// Mitsubishi GX Works2 project: 미쯔비시   PLC: Q02U

PROGRAM INPUT
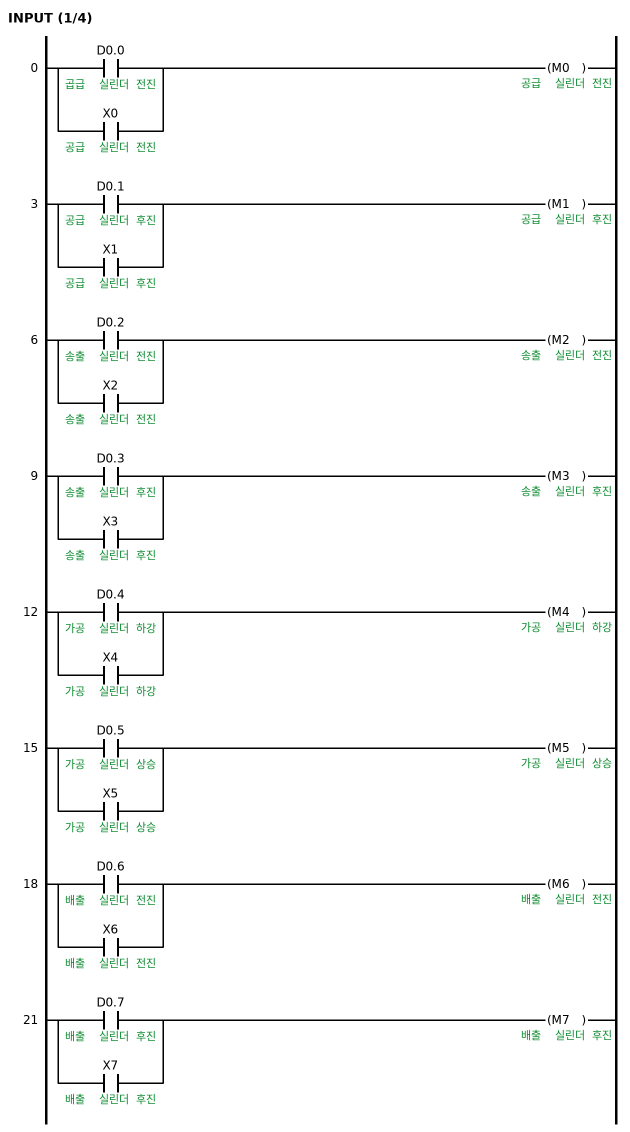
0     LD      D0.0  ; 곱급    실린더  전진
      OR      X0  ; 공급    실린더  전진
      OUT     M0  ; 공급    실린더  전진
3     LD      D0.1  ; 공급    실린더  후진
      OR      X1  ; 공급    실린더  후진
      OUT     M1  ; 공급    실린더  후진
6     LD      D0.2  ; 송출    실린더  전진
      OR      X2  ; 송출    실린더  전진
      OUT     M2  ; 송출    실린더  전진
9     LD      D0.3  ; 송출    실린더  후진
      OR      X3  ; 송출    실린더  후진
      OUT     M3  ; 송출    실린더  후진
12    LD      D0.4  ; 가공    실린더  하강
      OR      X4  ; 가공    실린더  하강
      OUT     M4  ; 가공    실린더  하강
15    LD      D0.5  ; 가공    실린더  상승
      OR      X5  ; 가공    실린더  상승
      OUT     M5  ; 가공    실린더  상승
18    LD      D0.6  ; 배출    실린더  전진
      OR      X6  ; 배출    실린더  전진
      OUT     M6  ; 배출    실린더  전진
21    LD      D0.7  ; 배출    실린더  후진
      OR      X7  ; 배출    실린더  후진
      OUT     M7  ; 배출    실린더  후진
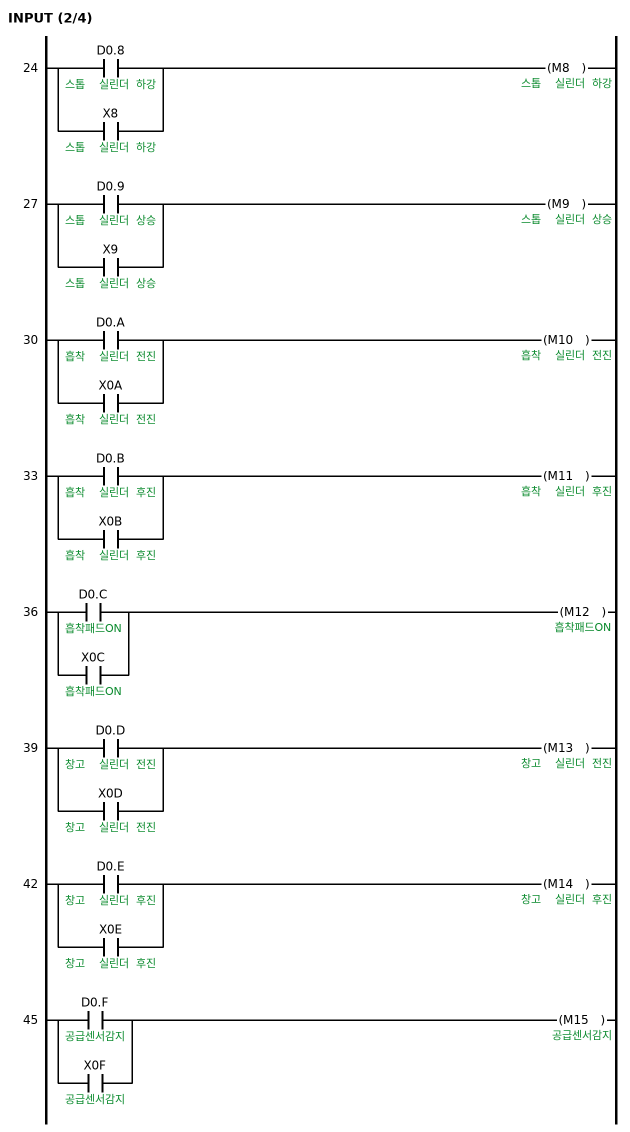
24    LD      D0.8  ; 스톱    실린더  하강
      OR      X8  ; 스톱    실린더  하강
      OUT     M8  ; 스톱    실린더  하강
27    LD      D0.9  ; 스톱    실린더  상승
      OR      X9  ; 스톱    실린더  상승
      OUT     M9  ; 스톱    실린더  상승
30    LD      D0.A  ; 흡착    실린더  전진
      OR      X0A  ; 흡착    실린더  전진
      OUT     M10  ; 흡착    실린더  전진
33    LD      D0.B  ; 흡착    실린더  후진
      OR      X0B  ; 흡착    실린더  후진
      OUT     M11  ; 흡착    실린더  후진
36    LD      D0.C  ; 흡착패드ON
      OR      X0C  ; 흡착패드ON
      OUT     M12  ; 흡착패드ON
39    LD      D0.D  ; 창고    실린더  전진
      OR      X0D  ; 창고    실린더  전진
      OUT     M13  ; 창고    실린더  전진
42    LD      D0.E  ; 창고    실린더  후진
      OR      X0E  ; 창고    실린더  후진
      OUT     M14  ; 창고    실린더  후진
45    LD      D0.F  ; 공급센서감지
      OR      X0F  ; 공급센서감지
      OUT     M15  ; 공급센서감지
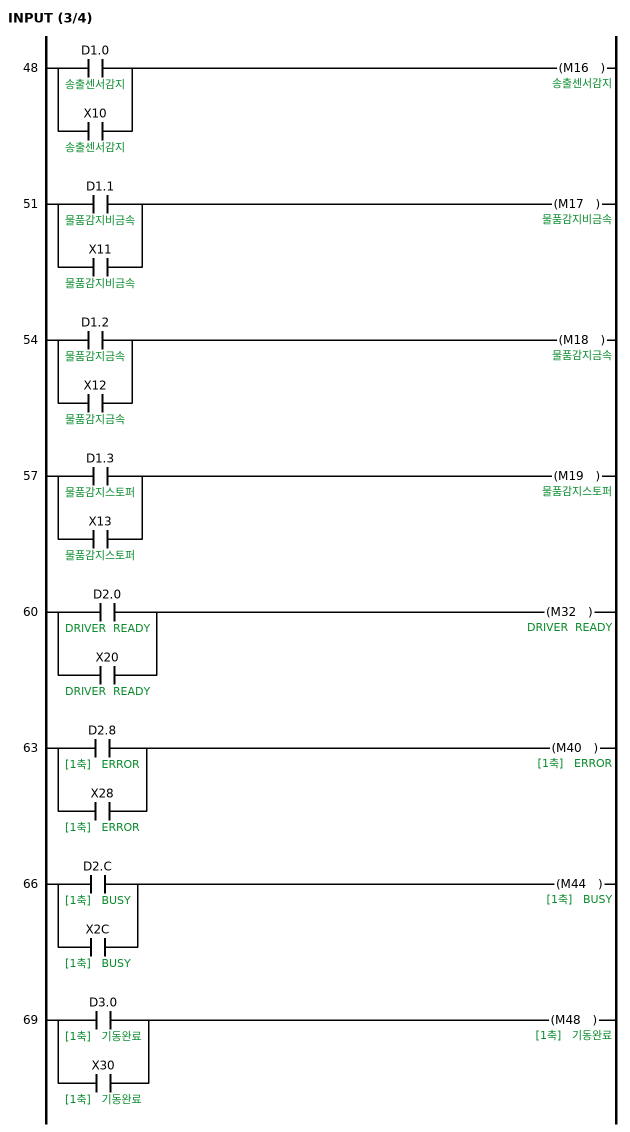
48    LD      D1.0  ; 송출센서감지
      OR      X10  ; 송출센서감지
      OUT     M16  ; 송출센서감지
51    LD      D1.1  ; 물품감지비금속
      OR      X11  ; 물품감지비금속
      OUT     M17  ; 물품감지비금속
54    LD      D1.2  ; 물품감지금속
      OR      X12  ; 물품감지금속
      OUT     M18  ; 물품감지금속
57    LD      D1.3  ; 물품감지스토퍼
      OR      X13  ; 물품감지스토퍼
      OUT     M19  ; 물품감지스토퍼
60    LD      D2.0  ; DRIVER  READY
      OR      X20  ; DRIVER  READY
      OUT     M32  ; DRIVER  READY
63    LD      D2.8  ; [1축]   ERROR
      OR      X28  ; [1축]   ERROR
      OUT     M40  ; [1축]   ERROR
66    LD      D2.C  ; [1축]   BUSY
      OR      X2C  ; [1축]   BUSY
      OUT     M44  ; [1축]   BUSY
69    LD      D3.0  ; [1축]   기동완료
      OR      X30  ; [1축]   기동완료
      OUT     M48  ; [1축]   기동완료
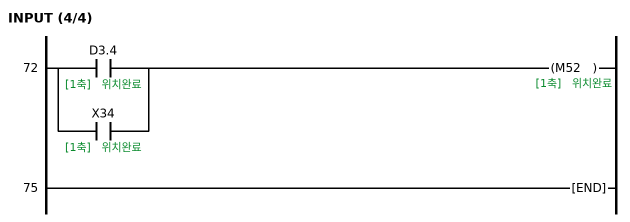
72    LD      D3.4  ; [1축]   위치완료
      OR      X34  ; [1축]   위치완료
      OUT     M52  ; [1축]   위치완료
75    END
END_PROGRAM

PROGRAM OUTPUT
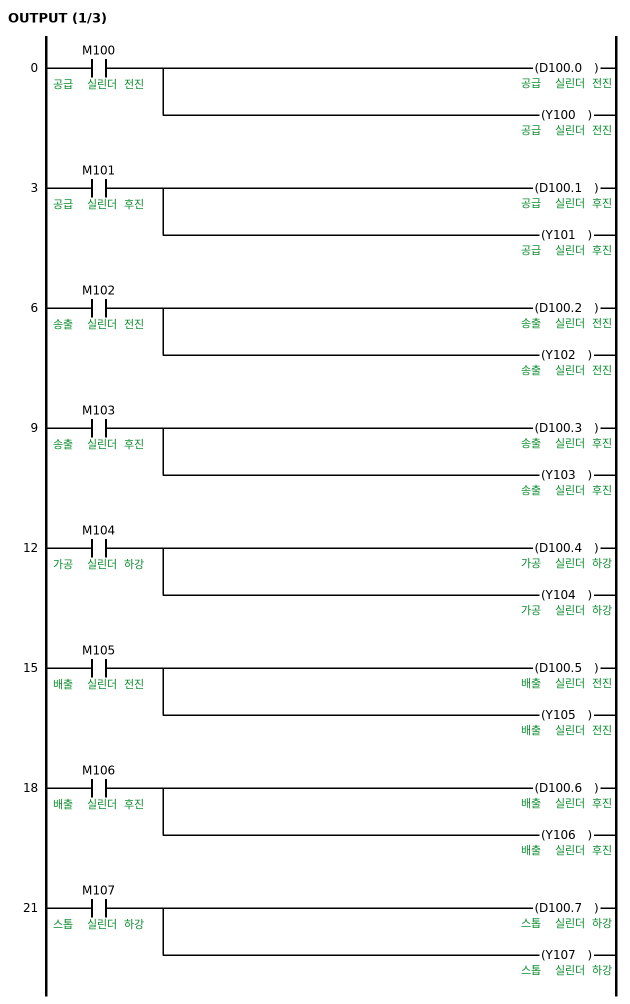
0     LD      M100  ; 공급    실린더  전진
      OUT     D100.0  ; 공급    실린더  전진
      OUT     Y100  ; 공급    실린더  전진
3     LD      M101  ; 공급    실린더  후진
      OUT     D100.1  ; 공급    실린더  후진
      OUT     Y101  ; 공급    실린더  후진
6     LD      M102  ; 송출    실린더  전진
      OUT     D100.2  ; 송출    실린더  전진
      OUT     Y102  ; 송출    실린더  전진
9     LD      M103  ; 송출    실린더  후진
      OUT     D100.3  ; 송출    실린더  후진
      OUT     Y103  ; 송출    실린더  후진
12    LD      M104  ; 가공    실린더  하강
      OUT     D100.4  ; 가공    실린더  하강
      OUT     Y104  ; 가공    실린더  하강
15    LD      M105  ; 배출    실린더  전진
      OUT     D100.5  ; 배출    실린더  전진
      OUT     Y105  ; 배출    실린더  전진
18    LD      M106  ; 배출    실린더  후진
      OUT     D100.6  ; 배출    실린더  후진
      OUT     Y106  ; 배출    실린더  후진
21    LD      M107  ; 스톱    실린더  하강
      OUT     D100.7  ; 스톱    실린더  하강
      OUT     Y107  ; 스톱    실린더  하강
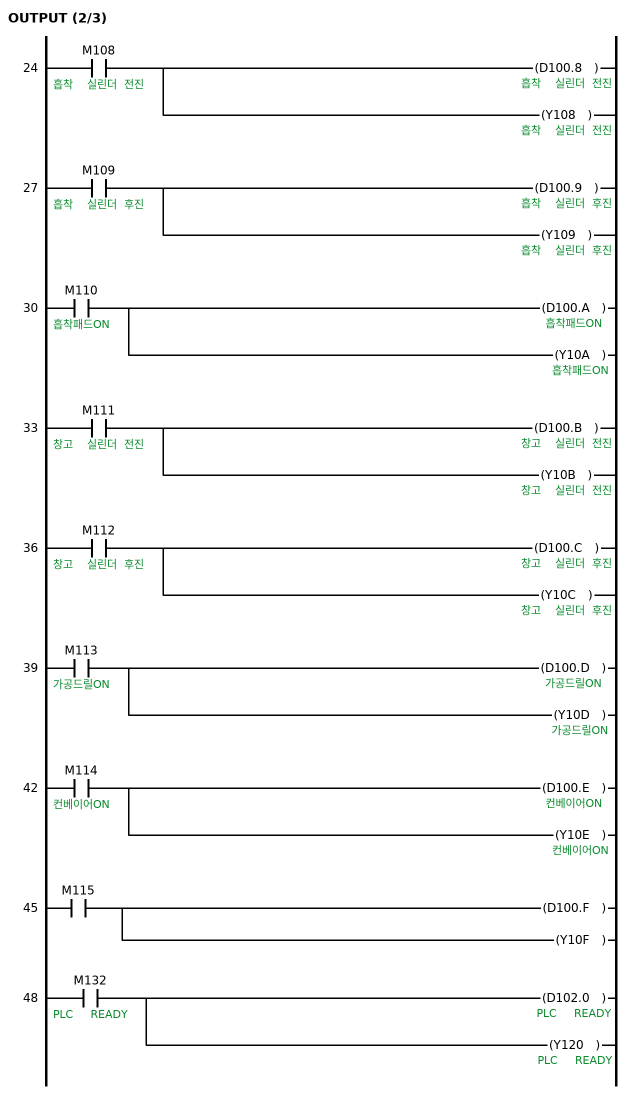
24    LD      M108  ; 흡착    실린더  전진
      OUT     D100.8  ; 흡착    실린더  전진
      OUT     Y108  ; 흡착    실린더  전진
27    LD      M109  ; 흡착    실린더  후진
      OUT     D100.9  ; 흡착    실린더  후진
      OUT     Y109  ; 흡착    실린더  후진
30    LD      M110  ; 흡착패드ON
      OUT     D100.A  ; 흡착패드ON
      OUT     Y10A  ; 흡착패드ON
33    LD      M111  ; 창고    실린더  전진
      OUT     D100.B  ; 창고    실린더  전진
      OUT     Y10B  ; 창고    실린더  전진
36    LD      M112  ; 창고    실린더  후진
      OUT     D100.C  ; 창고    실린더  후진
      OUT     Y10C  ; 창고    실린더  후진
39    LD      M113  ; 가공드릴ON
      OUT     D100.D  ; 가공드릴ON
      OUT     Y10D  ; 가공드릴ON
42    LD      M114  ; 컨베이어ON
      OUT     D100.E  ; 컨베이어ON
      OUT     Y10E  ; 컨베이어ON
45    LD      M115
      OUT     D100.F
      OUT     Y10F
48    LD      M132  ; PLC     READY
      OUT     D102.0  ; PLC     READY
      OUT     Y120  ; PLC     READY
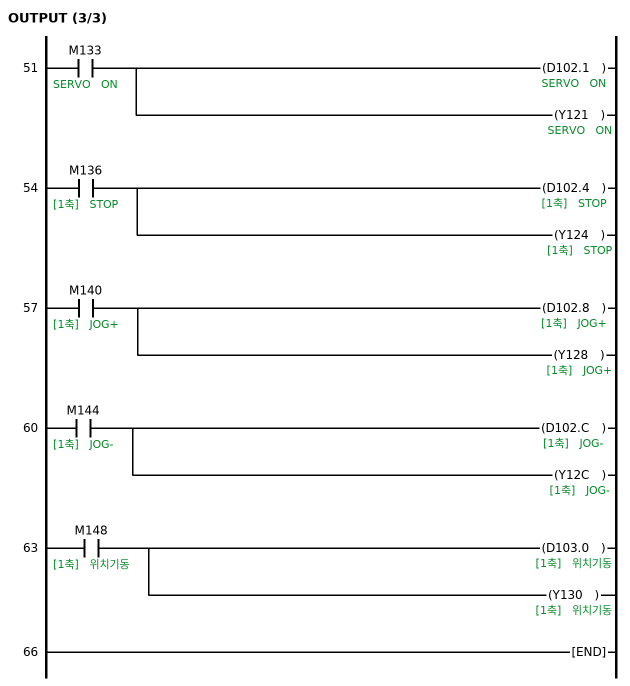
51    LD      M133  ; SERVO   ON
      OUT     D102.1  ; SERVO   ON
      OUT     Y121  ; SERVO   ON
54    LD      M136  ; [1축]   STOP
      OUT     D102.4  ; [1축]   STOP
      OUT     Y124  ; [1축]   STOP
57    LD      M140  ; [1축]   JOG+
      OUT     D102.8  ; [1축]   JOG+
      OUT     Y128  ; [1축]   JOG+
60    LD      M144  ; [1축]   JOG-
      OUT     D102.C  ; [1축]   JOG-
      OUT     Y12C  ; [1축]   JOG-
63    LD      M148  ; [1축]   위치기동
      OUT     D103.0  ; [1축]   위치기동
      OUT     Y130  ; [1축]   위치기동
66    END
END_PROGRAM

PROGRAM CONTROL
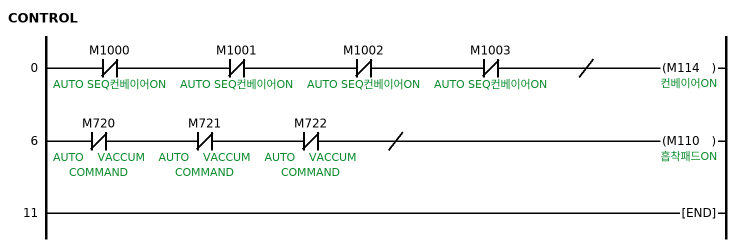
0     LDI     M1000  ; AUTO SEQ컨베이어ON
      ANI     M1001  ; AUTO SEQ컨베이어ON
      ANI     M1002  ; AUTO SEQ컨베이어ON
      ANI     M1003  ; AUTO SEQ컨베이어ON
      INV
      OUT     M114  ; 컨베이어ON
6     LDI     M720  ; AUTO    VACCUM  COMMAND
      ANI     M721  ; AUTO    VACCUM  COMMAND
      ANI     M722  ; AUTO    VACCUM  COMMAND
      INV
      OUT     M110  ; 흡착패드ON
11    END
END_PROGRAM

PROGRAM SUPPLY
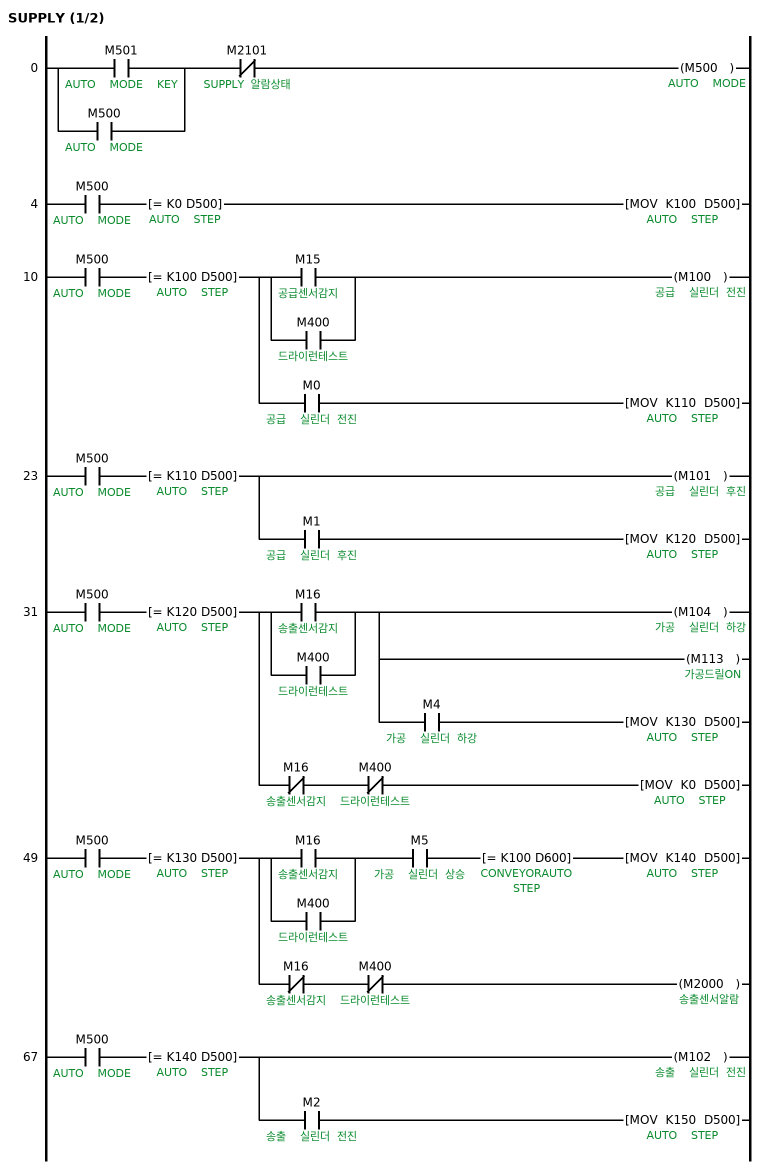
0     LD      M501  ; AUTO    MODE    KEY
      OR      M500  ; AUTO    MODE
      ANI     M2101  ; SUPPLY  알람상태
      OUT     M500  ; AUTO    MODE
4     LD      M500  ; AUTO    MODE
      AND=    K0 D500  ; AUTO    STEP
      MOV     K100 D500
10    LD      M500  ; AUTO    MODE
      AND=    K100 D500  ; AUTO    STEP
      MPS
      LD      M15  ; 공급센서감지
      OR      M400  ; 드라이런테스트
      ANB
      OUT     M100  ; 공급    실린더  전진
      MPP
      AND     M0  ; 공급    실린더  전진
      MOV     K110 D500
23    LD      M500  ; AUTO    MODE
      AND=    K110 D500  ; AUTO    STEP
      OUT     M101  ; 공급    실린더  후진
      AND     M1  ; 공급    실린더  후진
      MOV     K120 D500
31    LD      M500  ; AUTO    MODE
      AND=    K120 D500  ; AUTO    STEP
      MPS
      LD      M16  ; 송출센서감지
      OR      M400  ; 드라이런테스트
      ANB
      OUT     M104  ; 가공    실린더  하강
      OUT     M113  ; 가공드릴ON
      AND     M4  ; 가공    실린더  하강
      MOV     K130 D500
      MPP
      ANI     M16  ; 송출센서감지
      ANI     M400  ; 드라이런테스트
      MOV     K0 D500
49    LD      M500  ; AUTO    MODE
      AND=    K130 D500  ; AUTO    STEP
      MPS
      LD      M16  ; 송출센서감지
      OR      M400  ; 드라이런테스트
      ANB
      AND     M5  ; 가공    실린더  상승
      AND=    K100 D600  ; CONVEYORAUTO    STEP
      MOV     K140 D500
      MPP
      ANI     M16  ; 송출센서감지
      ANI     M400  ; 드라이런테스트
      OUT     M2000  ; 송출센서알람
67    LD      M500  ; AUTO    MODE
      AND=    K140 D500  ; AUTO    STEP
      OUT     M102  ; 송출    실린더  전진
      AND     M2  ; 송출    실린더  전진
      MOV     K150 D500
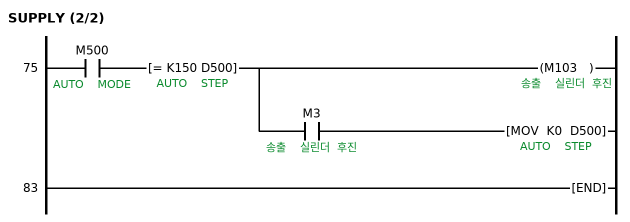
75    LD      M500  ; AUTO    MODE
      AND=    K150 D500  ; AUTO    STEP
      OUT     M103  ; 송출    실린더  후진
      AND     M3  ; 송출    실린더  후진
      MOV     K0 D500
83    END
END_PROGRAM

PROGRAM CONVEYOR
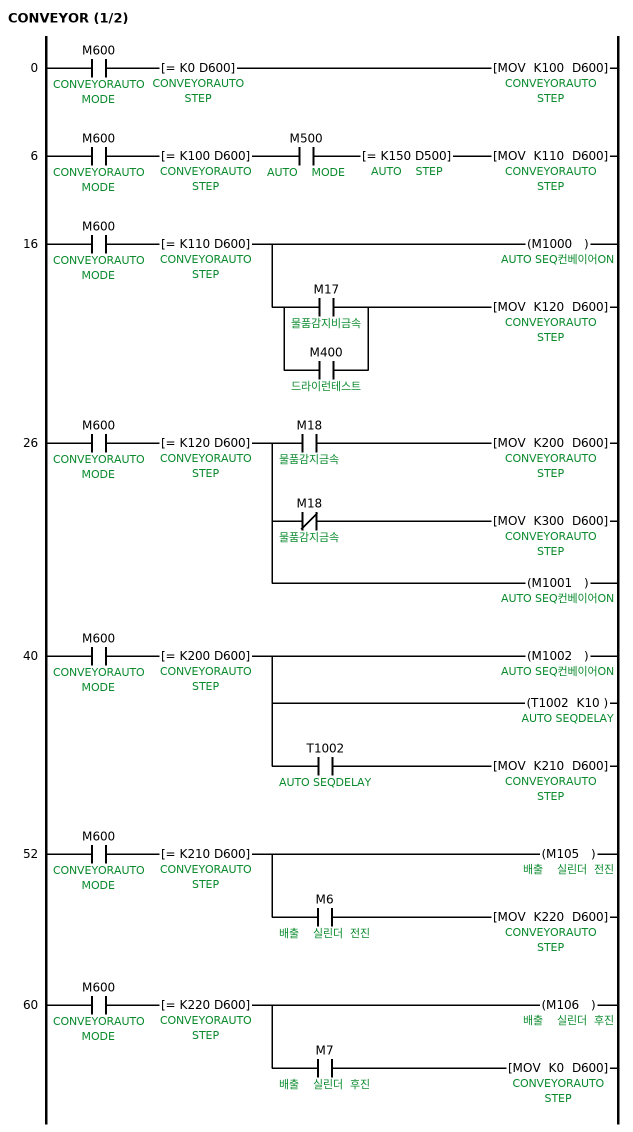
0     LD      M600  ; CONVEYORAUTO    MODE
      AND=    K0 D600  ; CONVEYORAUTO    STEP
      MOV     K100 D600
6     LD      M600  ; CONVEYORAUTO    MODE
      AND=    K100 D600  ; CONVEYORAUTO    STEP
      AND     M500  ; AUTO    MODE
      AND=    K150 D500  ; AUTO    STEP
      MOV     K110 D600
16    LD      M600  ; CONVEYORAUTO    MODE
      AND=    K110 D600  ; CONVEYORAUTO    STEP
      OUT     M1000  ; AUTO SEQ컨베이어ON
      LD      M17  ; 물품감지비금속
      OR      M400  ; 드라이런테스트
      ANB
      MOV     K120 D600
26    LD      M600  ; CONVEYORAUTO    MODE
      AND=    K120 D600  ; CONVEYORAUTO    STEP
      MPS
      AND     M18  ; 물품감지금속
      MOV     K200 D600
      MRD
      ANI     M18  ; 물품감지금속
      MOV     K300 D600
      MPP
      OUT     M1001  ; AUTO SEQ컨베이어ON
40    LD      M600  ; CONVEYORAUTO    MODE
      AND=    K200 D600  ; CONVEYORAUTO    STEP
      OUT     M1002  ; AUTO SEQ컨베이어ON
      OUT     T1002 K10  ; AUTO SEQDELAY
      AND     T1002  ; AUTO SEQDELAY
      MOV     K210 D600
52    LD      M600  ; CONVEYORAUTO    MODE
      AND=    K210 D600  ; CONVEYORAUTO    STEP
      OUT     M105  ; 배출    실린더  전진
      AND     M6  ; 배출    실린더  전진
      MOV     K220 D600
60    LD      M600  ; CONVEYORAUTO    MODE
      AND=    K220 D600  ; CONVEYORAUTO    STEP
      OUT     M106  ; 배출    실린더  후진
      AND     M7  ; 배출    실린더  후진
      MOV     K0 D600
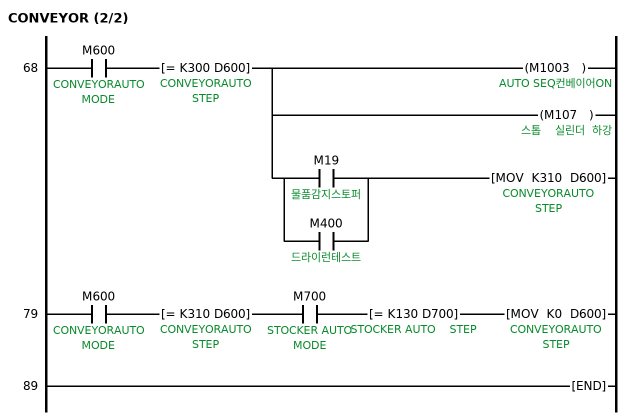
68    LD      M600  ; CONVEYORAUTO    MODE
      AND=    K300 D600  ; CONVEYORAUTO    STEP
      OUT     M1003  ; AUTO SEQ컨베이어ON
      OUT     M107  ; 스톱    실린더  하강
      LD      M19  ; 물품감지스토퍼
      OR      M400  ; 드라이런테스트
      ANB
      MOV     K310 D600
79    LD      M600  ; CONVEYORAUTO    MODE
      AND=    K310 D600  ; CONVEYORAUTO    STEP
      AND     M700  ; STOCKER AUTO    MODE
      AND=    K130 D700  ; STOCKER AUTO    STEP
      MOV     K0 D600
89    END
END_PROGRAM

PROGRAM STOCKER
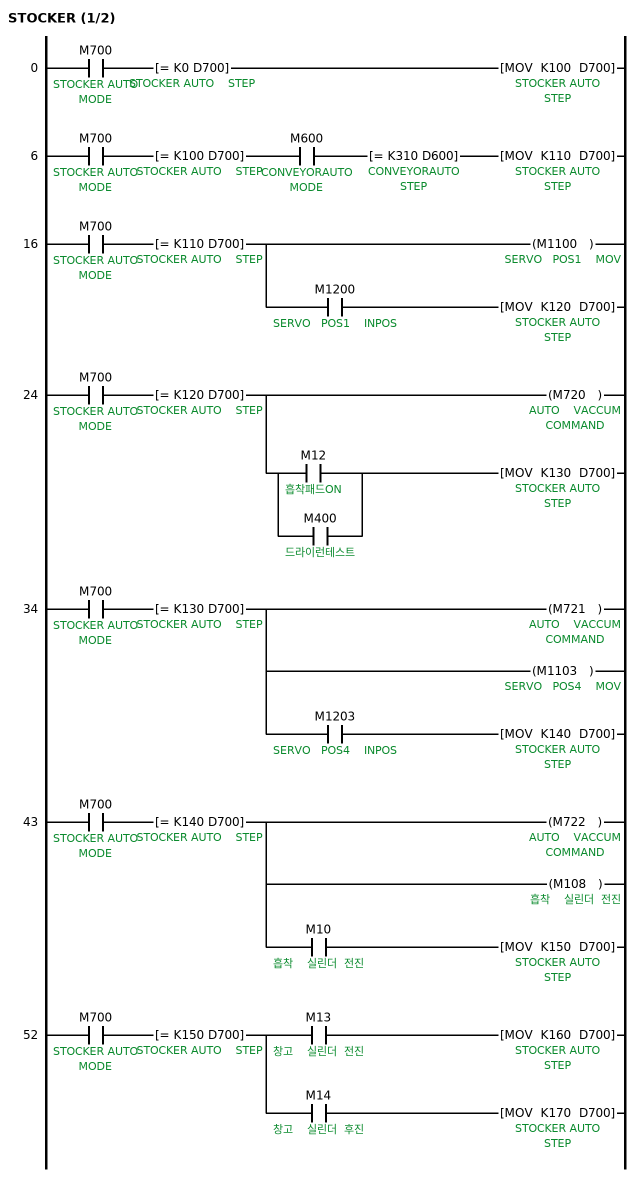
0     LD      M700  ; STOCKER AUTO    MODE
      AND=    K0 D700  ; STOCKER AUTO    STEP
      MOV     K100 D700
6     LD      M700  ; STOCKER AUTO    MODE
      AND=    K100 D700  ; STOCKER AUTO    STEP
      AND     M600  ; CONVEYORAUTO    MODE
      AND=    K310 D600  ; CONVEYORAUTO    STEP
      MOV     K110 D700
16    LD      M700  ; STOCKER AUTO    MODE
      AND=    K110 D700  ; STOCKER AUTO    STEP
      OUT     M1100  ; SERVO   POS1    MOV
      AND     M1200  ; SERVO   POS1    INPOS
      MOV     K120 D700
24    LD      M700  ; STOCKER AUTO    MODE
      AND=    K120 D700  ; STOCKER AUTO    STEP
      OUT     M720  ; AUTO    VACCUM  COMMAND
      LD      M12  ; 흡착패드ON
      OR      M400  ; 드라이런테스트
      ANB
      MOV     K130 D700
34    LD      M700  ; STOCKER AUTO    MODE
      AND=    K130 D700  ; STOCKER AUTO    STEP
      OUT     M721  ; AUTO    VACCUM  COMMAND
      OUT     M1103  ; SERVO   POS4    MOV
      AND     M1203  ; SERVO   POS4    INPOS
      MOV     K140 D700
43    LD      M700  ; STOCKER AUTO    MODE
      AND=    K140 D700  ; STOCKER AUTO    STEP
      OUT     M722  ; AUTO    VACCUM  COMMAND
      OUT     M108  ; 흡착    실린더  전진
      AND     M10  ; 흡착    실린더  전진
      MOV     K150 D700
52    LD      M700  ; STOCKER AUTO    MODE
      AND=    K150 D700  ; STOCKER AUTO    STEP
      MPS
      AND     M13  ; 창고    실린더  전진
      MOV     K160 D700
      MPP
      AND     M14  ; 창고    실린더  후진
      MOV     K170 D700
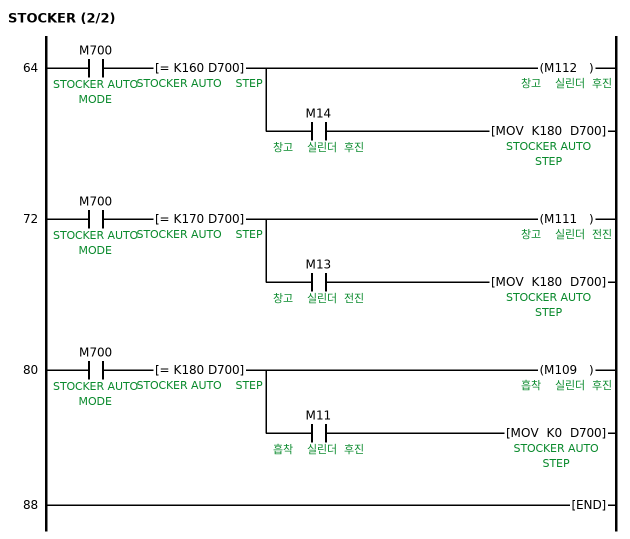
64    LD      M700  ; STOCKER AUTO    MODE
      AND=    K160 D700  ; STOCKER AUTO    STEP
      OUT     M112  ; 창고    실린더  후진
      AND     M14  ; 창고    실린더  후진
      MOV     K180 D700
72    LD      M700  ; STOCKER AUTO    MODE
      AND=    K170 D700  ; STOCKER AUTO    STEP
      OUT     M111  ; 창고    실린더  전진
      AND     M13  ; 창고    실린더  전진
      MOV     K180 D700
80    LD      M700  ; STOCKER AUTO    MODE
      AND=    K180 D700  ; STOCKER AUTO    STEP
      OUT     M109  ; 흡착    실린더  후진
      AND     M11  ; 흡착    실린더  후진
      MOV     K0 D700
88    END
END_PROGRAM

PROGRAM SERVO
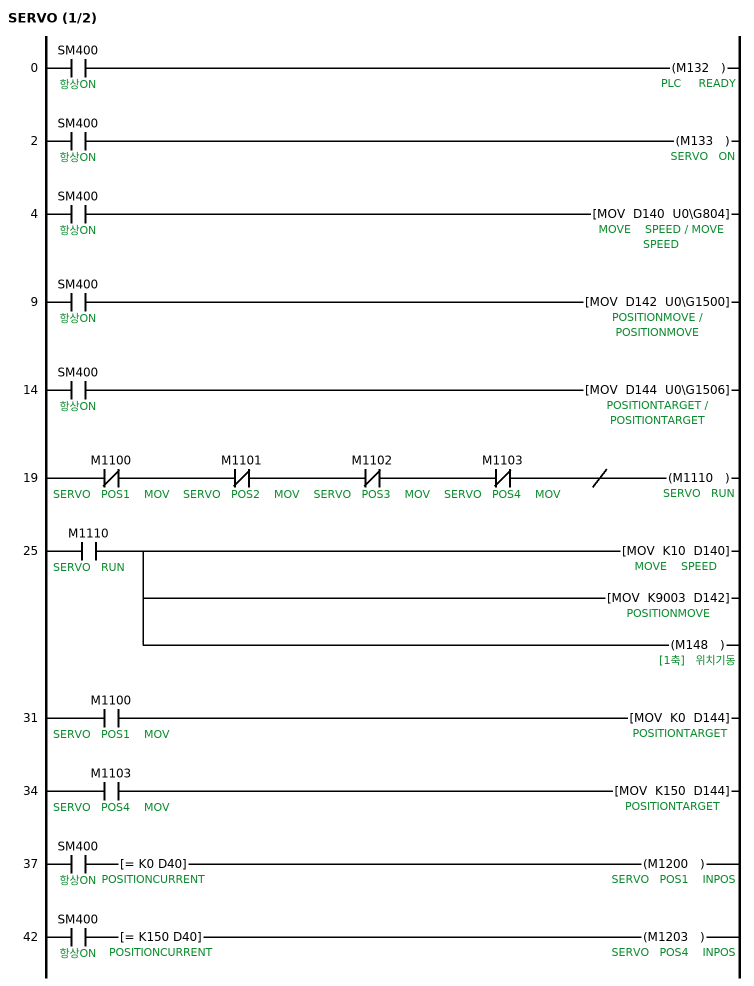
0     LD      SM400  ; 항상ON
      OUT     M132  ; PLC     READY
2     LD      SM400  ; 항상ON
      OUT     M133  ; SERVO   ON
4     LD      SM400  ; 항상ON
      MOV     D140 U0\G804  ; MOVE    SPEED / MOVE    SPEED
9     LD      SM400  ; 항상ON
      MOV     D142 U0\G1500  ; POSITIONMOVE / POSITIONMOVE
14    LD      SM400  ; 항상ON
      MOV     D144 U0\G1506  ; POSITIONTARGET / POSITIONTARGET
19    LDI     M1100  ; SERVO   POS1    MOV
      ANI     M1101  ; SERVO   POS2    MOV
      ANI     M1102  ; SERVO   POS3    MOV
      ANI     M1103  ; SERVO   POS4    MOV
      INV
      OUT     M1110  ; SERVO   RUN
25    LD      M1110  ; SERVO   RUN
      MOV     K10 D140
      MOV     K9003 D142
      OUT     M148  ; [1축]   위치기동
31    LD      M1100  ; SERVO   POS1    MOV
      MOV     K0 D144
34    LD      M1103  ; SERVO   POS4    MOV
      MOV     K150 D144
37    LD      SM400  ; 항상ON
      AND=    K0 D40  ; POSITIONCURRENT
      OUT     M1200  ; SERVO   POS1    INPOS
42    LD      SM400  ; 항상ON
      AND=    K150 D40  ; POSITIONCURRENT
      OUT     M1203  ; SERVO   POS4    INPOS
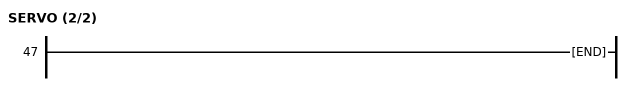
47    END
END_PROGRAM

PROGRAM ALARM
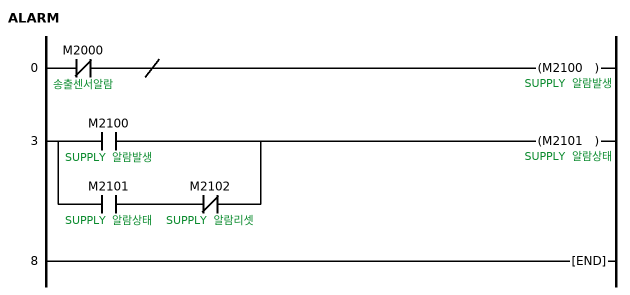
0     LDI     M2000  ; 송출센서알람
      INV
      OUT     M2100  ; SUPPLY  알람발생
3     LD      M2100  ; SUPPLY  알람발생
      LD      M2101  ; SUPPLY  알람상태
      ANI     M2102  ; SUPPLY  알람리셋
      ORB
      OUT     M2101  ; SUPPLY  알람상태
8     END
END_PROGRAM

// device comments not shown above
M199  ; SIMUL   MODE
